PROGRAM MAIN
VAR
    TestSuite_AssertTests : TestSuite_AssertTests;
    TestSuite_ListOfTests : TestSuite_ListOfTests;
END_VAR

TestSuite_AssertTests();
TestSuite_ListOfTests();

END_PROGRAM

(* stored: Version 1.1.0.1, ProductVersion 3.1.4024.12
   POU MAIN: Id {cfaff396-02d6-4fc1-bf48-96a5a0da3de0}, SpecialFunc None *)
